// TIA Portal V17 export
FUNCTION "FC_BurnerAlarm" : Void   // FC, LAD
{ S7_Optimized_Access := 'TRUE' }
BEGIN
END_FUNCTION
